{attribute 'qualified_only'}
VAR_GLOBAL CONSTANT
    MaxHandlers : DINT := 5;
END_VAR

(* stored: Version 1.1.0.1, ProductVersion 3.1.4024.3
   GVL Parameters: Id {dd27dcd6-341e-49c9-9aa0-10b2802af1ee}, ParameterList True *)
